# B&R Automation Studio project Sew
Automation Studio 4.9

## Configuration Config1

### Task classes (Cpu.sw)
```
Cyclic#4:
  Test <- Test.prg
```

## Logical view

### Program Logical/Test

#### Main.st
```iecst
PROGRAM _INIT
	(* Insert code here *)

END_PROGRAM

PROGRAM _CYCLIC
	(* Insert code here *)
	IF Test THEN
		Test := 1;
	END_IF;
END_PROGRAM

PROGRAM _EXIT
	(* Insert code here *)

END_PROGRAM
```
